(* IEC 61131-3 sources: Industry-PLC-LLM/data/PLCBEAD_repo/PLCBEAD_PLCEmbed-main/PLC-BEAD/Source/GEB/CARG, 1 file *)

(* ---- CARG.ST ---- *)
TYPE oscat_complex :
  STRUCT
	re : REAL;
	im : REAL;
  END_STRUCT;
END_TYPE

FUNCTION ATAN2:REAL
	VAR_INPUT
		X :	REAL;
		Y :	REAL;
	END_VAR

	IF X > 0.0 THEN
		ATAN2 := ATAN(Y/X);
	ELSIF X < 0.0 THEN
		IF Y >= 0.0 THEN
			ATAN2 := ATAN(Y/X) + 3.14159265358979323846264338327950288;
		ELSE
			ATAN2 := ATAN(Y/X) - 3.14159265358979323846264338327950288;
		END_IF;
	ELSIF Y > 0.0 THEN
		ATAN2 := 1.5707963267948965580;
	ELSIF Y < 0.0 THEN
		ATAN2 := -1.5707963267948965580;
	ELSE
		ATAN2 := 0.0;
	END_IF;

END_FUNCTION

FUNCTION_BLOCK CARG_Block

	VAR_INPUT
		X :	oscat_complex;
	END_VAR

	VAR_OUTPUT
		CARG :	REAL;
	END_VAR

	CARG := ATAN2(X.im, X.re);

END_FUNCTION_BLOCK

PROGRAM program0
  VAR
    LocalVar0 : oscat_complex;
	LocalOUT  : REAL;
	func_block : CARG_Block;
  END_VAR
	func_block.X  := LocalVar0;
	func_block();
	LocalOUT := func_block.CARG;
END_PROGRAM
